FUNCTION_BLOCK E_D_FF_ANY_1 (* Data latch (d) flip flop for 1 ANY variable, EO only on change of at least one Q (generic FB) *)
  (* Standard: 61499-1 Annex A; Description: Copyright (c) 2017, 2026 fortiss GmbH, HR Agrartechnik GmbH This program and the accompanying materials are made available under the terms of the Eclipse Public License 2.0 which is available at https://www.eclipse.org/legal/epl-2.0/ SPDX-License-Identifier: EPL-2.0 *)
  (* Version 1.0, 2026-08-26, Franz Höpfinger, HR Agrartechnik GmbH, E_D_FF_ANY extended to 1 variable - EO fires only if at least one Di differs from the latched Qi. Service Interface FB, native implementation GEN_E_D_FF_ANY (FORTE) required. *)
  PACKAGE iec61499::events;
  {SET_ATTRIBUTE(eclipse4diac::core::GenericClassName, 'GEN_E_D_FF_ANY')}
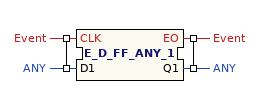
  EVENT_INPUT
    CLK WITH D1; (* Clock *)
  END_EVENT
  EVENT_OUTPUT
    EO WITH Q1; (* Triggered if clock results in a change of at least one Q *)
  END_EVENT
  VAR_INPUT
    D1 : ANY; (* Value 1 to latch *)
  END_VAR
  VAR_OUTPUT
    Q1 : ANY; (* Latched value 1 *)
  END_VAR
END_FUNCTION_BLOCK
